TYPE Warning_FLC_DINT :
UNION
	Value : DINT;
	Bits  : Warnings_FLC;
END_UNION
END_TYPE

(* stored: Version 1.1.0.1, ProductVersion 3.1.4024.4
   DUT Warning_FLC_DINT: Id {d1142580-c5fb-4edb-a3ea-206f7a85d711} *)
